{attribute addProperty BoxType ""}
{attribute addProperty Id "unreferencedAT %I*SyncUnitTask_B4157F22658.1250PlcTaskAT %I*SyncUnitTask_B4157F22658.1250PlcTask1AT %I*SyncUnitTask_B4157F22658.1250"}
{attribute addProperty CRC "1214597596"}
{attribute addProperty SizeInBites "195"}
{attribute addProperty SizeInBytes "24.375"}
TYPE SyncUnitTasks_486549DC :
STRUCT
	{attribute addProperty Name "unreferenced"}
	unreferenced : SyncUnitTask_B4157F22;
	{attribute addProperty Name "PlcTask"}
	PlcTask : SyncUnitTask_B4157F22;
	{attribute addProperty Name "PlcTask1"}
	PlcTask1 : SyncUnitTask_B4157F22;
END_STRUCT
END_TYPE

(* stored: Version 1.2.0.0, ProductVersion 3.1.4024.9
   DUT SyncUnitTasks_486549DC: Id {9b828ea2-cd00-4138-9d0d-3ebab5915345} *)
